(* IEC 61131-3 sources: POMIRTS_lab3/AS/Library/AsIO, 2 files *)

(* ---- AsIO.fun ---- *)
(********************************************************************
 * COPYRIGHT -- Bernecker + Rainer
 ********************************************************************
 * Library: AsIO
 * File: AsIO.fun
 * Author: B+R
 ********************************************************************
 * Functions and function blocks of library AsIO
 ********************************************************************)

FUNCTION_BLOCK AsIODPStatus				(*determines the state and current value of an I/O data point; asynchronous execution*)
	VAR_INPUT
		enable       : BOOL; 			(*enables execution*)
		pDatapoint   : UDINT; 			(*I/O data point name given as a pointer*)
	END_VAR

	VAR
        i_state      : UINT;			(*internal variable*)
        i_result     : UINT;			(*internal variable*)
        unused       : UDINT;			(*internal variable*)
	END_VAR

	VAR_OUTPUT
		status       : UINT; 			(*execution status: ERR_OK, ERR_FUB_ENABLE_FALSE, ERR_FUB_BUSY, 0xXXXX = see help*)
        flags        : USINT;			(*information about the state of the data point*)
        datatype     : USINT;			(*data type of the data point according to the profibus standard*)
        value        : UDINT;			(*value of the data point*)
        forceValue   : UDINT;			(*force value of the data point*)
        defaultValue : UDINT;			(*default value of the data point*)
	END_VAR

END_FUNCTION_BLOCK

FUNCTION_BLOCK AsIOSetForceValue		(*sets the value of an I/O data point's "force" status; asynchronous execution*)
	VAR_INPUT
		enable       : BOOL; 			(*enables execution*)
		pDatapoint   : UDINT; 			(*I/O data point name given as a pointer*)
        value        : UDINT;			(*force value*)
	END_VAR

	VAR
        i_state      : UINT;			(*internal variable*)
        i_result     : UINT;			(*internal variable*)
        unused       : UDINT;			(*internal variable*)
	END_VAR

	VAR_OUTPUT
		status  : UINT; 				(*execution status: ERR_OK, ERR_FUB_ENABLE_FALSE, ERR_FUB_BUSY, 0xXXXX = see help*)
	END_VAR

END_FUNCTION_BLOCK

FUNCTION_BLOCK AsIOEnableForcing		(*enables the "force" status of an I/O data point; asynchronous execution*)
	VAR_INPUT
		enable       : BOOL; 			(*enables execution*)
		pDatapoint   : UDINT; 			(*I/O data point name given as a pointer*)
	END_VAR

	VAR
        i_state      : UINT;			(*internal variable*)
        i_result     : UINT;			(*internal variable*)
        unused       : UDINT;			(*internal variable*)
	END_VAR

	VAR_OUTPUT
		status  : UINT; 				(*execution status: ERR_OK, ERR_FUB_ENABLE_FALSE, ERR_FUB_BUSY, 0xXXXX = see help*)
	END_VAR

END_FUNCTION_BLOCK

FUNCTION_BLOCK AsIODisableForcing		(*disables the "force" status of an I/O data point; asynchronous execution*)
	VAR_INPUT
		enable       : BOOL; 			(*enables execution*)
		pDatapoint   : UDINT; 			(*I/O data point name given as a pointer*)
	END_VAR

	VAR
        i_state      : UINT;			(*internal variable*)
        i_result     : UINT;			(*internal variable*)
        unused       : UDINT;			(*internal variable*)
	END_VAR

	VAR_OUTPUT
		status  : UINT; 				(*execution status: ERR_OK, ERR_FUB_ENABLE_FALSE, ERR_FUB_BUSY, 0xXXXX = see help*)
	END_VAR

END_FUNCTION_BLOCK

FUNCTION_BLOCK AsIOGlobalDisableForcing	(*disables the "force" status of all I/O data points; asynchronous execution*)
	VAR_INPUT
		enable           : BOOL; 		(*enables execution*)
	END_VAR

	VAR
        i_state      : UINT;			(*internal variable*)
        i_result     : UINT;			(*internal variable*)
        unused       : UDINT;			(*internal variable*)
	END_VAR

	VAR_OUTPUT
		status  : UINT; 				(*execution status: ERR_OK, ERR_FUB_ENABLE_FALSE, ERR_FUB_BUSY, 0xXXXX = see help*)
	END_VAR

END_FUNCTION_BLOCK

FUNCTION_BLOCK AsIOListDP				(*determines the existing I/O data points; asynchronous execution*)
	VAR_INPUT
		enable       : BOOL; 			(*enables execution*)
		pLastDatapoint   : UDINT; 		(*old data point name given as a pointer*)
	END_VAR

	VAR
        i_state      : UINT;			(*internal variable*)
        i_result     : UINT;			(*internal variable*)
        unused       : UDINT;			(*internal variable*)
        buffer       : ARRAY[0..127] OF USINT;	(*internal variable*)
	END_VAR

	VAR_OUTPUT
		status       : UINT; 			(*execution status: ERR_OK, ERR_FUB_ENABLE_FALSE, ERR_FUB_BUSY, 0xXXXX = see help*)
		pDatapoint   : UDINT; 			(*data point name given as a pointer*)
	END_VAR

END_FUNCTION_BLOCK

FUNCTION_BLOCK AsIOPVInfo				(*collects data about PV's that are linked with a data point; asynchronous execution*)
   VAR_INPUT
       enable     : BOOL;				(*enables execution*)
       pDatapoint : UDINT;				(*I/O data point name given as a pointer*)
       index      : UDINT;				(*index of the searched PV*)
   END_VAR

   VAR
       i_state      : UINT;				(*internal variable*)
       i_result     : UINT;				(*internal variable*)
       bufferA       : ARRAY[0..127] OF USINT;	(*internal variable*)
       bufferB       : ARRAY[0..127] OF USINT;	(*internal variable*)
   END_VAR

	VAR_OUTPUT
		status       : UINT; 			(*execution status: ERR_OK, ERR_FUB_ENABLE_FALSE, ERR_FUB_BUSY, 0xXXXX = see help*)
		pPvName      : UDINT; 			(*PV names given as pointer, 0 if there is no PV linked with the specified index*)
		pPvContext   : UDINT; 			(*context names (given as a pointer) that are used to map this PV*)
        flags        : USINT;			(*additional information*)
	END_VAR

END_FUNCTION_BLOCK

(* ---- AsIO.var ---- *)
(********************************************************************
 * COPYRIGHT -- Bernecker + Rainer
 ********************************************************************
 * Library: AsIO
 * File: AsIO.var
 * Author: B+R
 ********************************************************************
 * Local variables of library AsIO
 ********************************************************************)

VAR CONSTANT
    asioERR_INTERNAL  : UINT := 30150;			(*internal error*)
    asioERR_NOSUCH_DP : UINT := 30151;			(*data point with specified name not found*)

    asio_VALID_FLAG         : USINT :=  1;		(*bit0 is always set*)
    asio_P_ACT_FLAG         : USINT :=  2;		(*bit1 = 1 data source active, bit1 = 0 data source inactive*)
    asio_F_ACT_FLAG         : USINT :=  4;		(*bit2 = 1 force active, bit2 = 0 force inactive*)
    asio_UNRES_LINK_FLAG    : USINT :=  8;		(*AsPVInfo: bit3=0 the PV link is established ,  AsIODPStatus: bit3=0 all PV links are established*)
    asio_IO_INPUT_FLAG      : USINT := 16;		(*the data point is an I/O input channel*)
    asio_IO_OUTPUT_FLAG     : USINT := 32;		(*the data point is an I/O output channel*)
	asio_IO_SIMULATION_FLAG : USINT := 64;      (*the data point is simulated*)
	asio_UNRES_IO_FLAG      : USINT :=128;      (*IO-Link unresolved*)

    asio_INVERTED_FLAG   : USINT := 64;			(*AsPVInfo:the PV link is inverted*)
END_VAR
